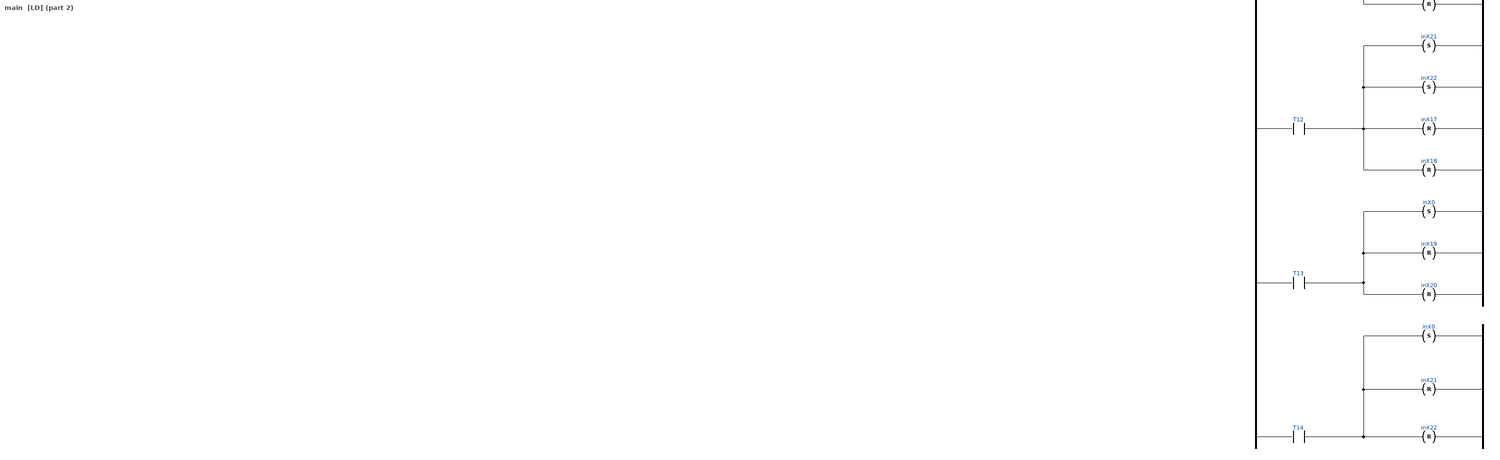
IF T12 THEN inX18 := FALSE; END_IF;
IF T12 THEN inX21 := TRUE; END_IF;
IF T12 THEN inX17 := FALSE; END_IF;
IF T12 THEN inX22 := TRUE; END_IF;
IF T13 THEN inX0 := TRUE; END_IF;
IF T13 THEN inX19 := FALSE; END_IF;
IF T13 THEN inX20 := FALSE; END_IF;
IF T14 THEN inX0 := TRUE; END_IF;
IF T14 THEN inX21 := FALSE; END_IF;
IF T14 THEN inX22 := FALSE; END_IF;
start := termX0;
_AND266_OUT := termX1 AND termX2 AND termX3;
WebGuide := _AND266_OUT;
CoilCar := _AND266_OUT;
Unwind := _AND266_OUT;
TensionSetup := termX4;
_AND271_OUT := termX5 AND termX6;
BottomKnife := _AND271_OUT;
TopKnife := _AND271_OUT;
_AND274_OUT := termX7 AND termX8;
MainDrive := _AND274_OUT;
PinchRoll := _AND274_OUT;
_AND277_OUT := termX9 AND termX10;
SlitWind := _AND277_OUT;
CoreShaft := _AND277_OUT;
_AND280_OUT := termX11 AND termX12;
NotchEdge := _AND280_OUT;
NotchUnwind := _AND280_OUT;
Press := termX15;
LaserSensor := termX16;
_AND287_OUT := termX19 AND termX20;
UnloadConv := _AND287_OUT;
Stack := _AND287_OUT;
_AND288_OUT := termX21 AND termX22;
RejConv := _AND288_OUT;
RejGate := _AND288_OUT;
BernoulliGenerator0(in := termX13 AND termX14, seed := seed_0);
Mechanical := BernoulliGenerator0.out_1;
Accum := BernoulliGenerator0.out_1 OR BernoulliGenerator0.out_2;
Laser := BernoulliGenerator0.out_2;
BernoulliGenerator1(in := termX17 AND termX18, seed := seed_1);
ElectrodePass := BernoulliGenerator1.out_1;
Vision := BernoulliGenerator1.out_1 OR BernoulliGenerator1.out_2;
ElectrodePass := NOT BernoulliGenerator1.out_2;
Dancer := BernoulliGenerator0.out_1 OR BernoulliGenerator0.out_2;
OQCConv := BernoulliGenerator1.out_1 OR BernoulliGenerator1.out_2;
END_PROGRAM

PROGRAM main2
  VAR
    inX0 : BOOL := TRUE;
    inX1 : BOOL;
    inX2 : BOOL;
    inX3 : BOOL;
    inX4 : BOOL;
    inX5 : BOOL;
    inX6 : BOOL;
    inX7 : BOOL;
    inX8 : BOOL;
    inX9 : BOOL;
    inX10 : BOOL;
    inX11 : BOOL;
    inX12 : BOOL;
    inX13 : BOOL;
    inX14 : BOOL;
    inX15 : BOOL;
    outX0 : BOOL;
    outX1 : BOOL;
    outX2 : BOOL;
    outX3 : BOOL;
    outX4 : BOOL;
    outX5 : BOOL;
    outX6 : BOOL;
    outX7 : BOOL;
    outX8 : BOOL;
    outX9 : BOOL;
    outX10 : BOOL;
    outX11 : BOOL;
    outX12 : BOOL;
    outX13 : BOOL;
    outX14 : BOOL;
    outX15 : BOOL;
    signalX0 : REAL;
    signalX1 : REAL;
    signalX2 : REAL;
    signalX3 : REAL;
    signalX4 : REAL;
    signalX5 : REAL;
    signalX6 : REAL;
    signalX7 : REAL;
    signalX8 : REAL;
    signalX9 : REAL;
    signalX10 : REAL;
    signalX11 : REAL;
    signalX12 : REAL;
    signalX13 : REAL;
    signalX14 : REAL;
    signalX15 : REAL;
    T0 : BOOL;
    T1 : BOOL;
    T2 : BOOL;
    T3 : BOOL;
    T4 : BOOL;
    T5 : BOOL;
    T6 : BOOL;
    T7 : BOOL;
    start : BOOL;
    ConvWeb : BOOL;
    TensWeb : BOOL;
    ConvCoat : BOOL;
    TensCoat : BOOL;
    PumpCoat : BOOL;
    ValveCoat : BOOL;
    ConvLevel : BOOL;
    TensLevel : BOOL;
    TensDryB : BOOL;
    AirB : BOOL;
    Heater : BOOL;
    AirA : BOOL;
    ConvQC : BOOL;
    TensQC : BOOL;
    Reset : BOOL;
    termX0 : BOOL;
    termX1 : BOOL;
    termX2 : BOOL;
    termX3 : BOOL;
    termX4 : BOOL;
    termX5 : BOOL;
    termX6 : BOOL;
    termX7 : BOOL;
    termX8 : BOOL;
    termX9 : BOOL;
    termX10 : BOOL;
    termX11 : BOOL;
    termX12 : BOOL;
    termX13 : BOOL;
    termX14 : BOOL;
    termX15 : BOOL;
    PVG0 : ProcessVariationGeneratorX0;
    PVG1 : ProcessVariationGeneratorX1;
    PVG2 : ProcessVariationGeneratorX2;
    PVG3 : ProcessVariationGeneratorX3;
    PVG4 : ProcessVariationGeneratorX4;
    PVG5 : ProcessVariationGeneratorX5;
    PVG6 : ProcessVariationGeneratorX6;
    PVG7 : ProcessVariationGeneratorX7;
    PVG8 : ProcessVariationGeneratorX8;
    PVG9 : ProcessVariationGeneratorX9;
    PVG10 : ProcessVariationGeneratorX10;
    PVG11 : ProcessVariationGeneratorX11;
    PVG12 : ProcessVariationGeneratorX12;
    PVG13 : ProcessVariationGeneratorX13;
    PVG14 : ProcessVariationGeneratorX14;
    PVG15 : ProcessVariationGeneratorX15;
  END_VAR

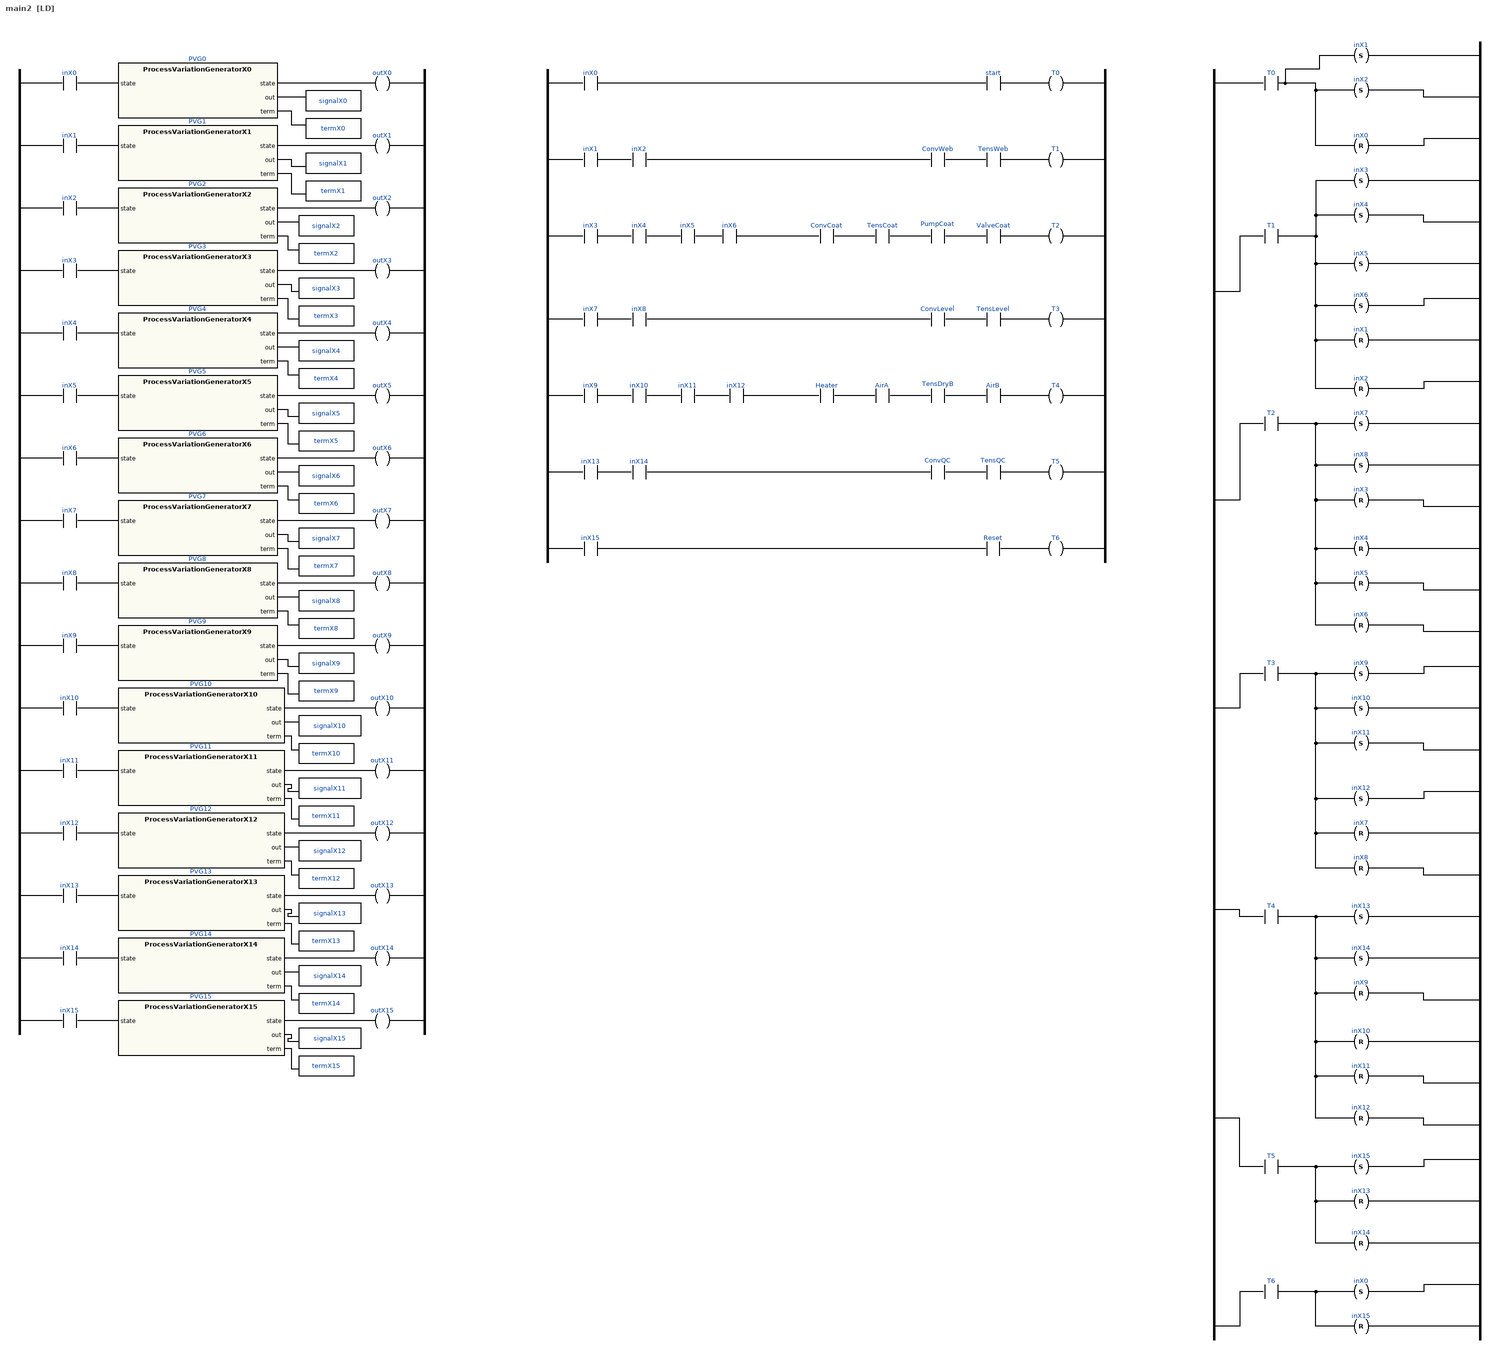
(* LD diagram, written out as Structured Text *)
PVG0(state := inX0);
outX0 := PVG0.state;
PVG1(state := inX1);
outX1 := PVG1.state;
PVG2(state := inX2);
outX2 := PVG2.state;
PVG3(state := inX3);
outX3 := PVG3.state;
PVG4(state := inX4);
outX4 := PVG4.state;
PVG5(state := inX5);
outX5 := PVG5.state;
PVG6(state := inX6);
outX6 := PVG6.state;
PVG7(state := inX7);
outX7 := PVG7.state;
PVG8(state := inX8);
outX8 := PVG8.state;
PVG9(state := inX9);
outX9 := PVG9.state;
PVG10(state := inX10);
outX10 := PVG10.state;
PVG11(state := inX11);
outX11 := PVG11.state;
PVG12(state := inX12);
outX12 := PVG12.state;
PVG13(state := inX13);
outX13 := PVG13.state;
PVG14(state := inX14);
outX14 := PVG14.state;
PVG15(state := inX15);
outX15 := PVG15.state;
signalX3 := PVG3.out;
signalX4 := PVG4.out;
signalX5 := PVG5.out;
signalX6 := PVG6.out;
signalX7 := PVG7.out;
signalX8 := PVG8.out;
signalX14 := PVG14.out;
signalX13 := PVG13.out;
signalX12 := PVG12.out;
signalX11 := PVG11.out;
signalX10 := PVG10.out;
signalX9 := PVG9.out;
signalX15 := PVG15.out;
signalX2 := PVG2.out;
signalX1 := PVG1.out;
signalX0 := PVG0.out;
T0 := inX0 AND start;
T1 := inX1 AND inX2 AND ConvWeb AND TensWeb;
T2 := inX3 AND inX4 AND inX5 AND inX6 AND ConvCoat AND TensCoat AND PumpCoat AND ValveCoat;
T3 := inX7 AND inX8 AND ConvLevel AND TensLevel;
T4 := inX9 AND inX10 AND inX11 AND inX12 AND Heater AND AirA AND TensDryB AND AirB;
T5 := inX13 AND inX14 AND ConvQC AND TensQC;
T6 := inX15 AND Reset;
IF T0 THEN inX1 := TRUE; END_IF;
IF T0 THEN inX2 := TRUE; END_IF;
IF T0 THEN inX0 := FALSE; END_IF;
IF T1 THEN inX3 := TRUE; END_IF;
IF T1 THEN inX4 := TRUE; END_IF;
IF T1 THEN inX5 := TRUE; END_IF;
IF T1 THEN inX6 := TRUE; END_IF;
IF T1 THEN inX1 := FALSE; END_IF;
IF T1 THEN inX2 := FALSE; END_IF;
IF T2 THEN inX8 := TRUE; END_IF;
IF T2 THEN inX3 := FALSE; END_IF;
IF T2 THEN inX4 := FALSE; END_IF;
IF T2 THEN inX5 := FALSE; END_IF;
IF T2 THEN inX6 := FALSE; END_IF;
IF T2 THEN inX7 := TRUE; END_IF;
IF T3 THEN inX9 := TRUE; END_IF;
IF T3 THEN inX10 := TRUE; END_IF;
IF T3 THEN inX11 := TRUE; END_IF;
IF T3 THEN inX12 := TRUE; END_IF;
IF T3 THEN inX7 := FALSE; END_IF;
IF T3 THEN inX8 := FALSE; END_IF;
IF T4 THEN inX13 := TRUE; END_IF;
IF T4 THEN inX14 := TRUE; END_IF;
IF T5 THEN inX13 := FALSE; END_IF;
IF T5 THEN inX14 := FALSE; END_IF;
IF T6 THEN inX0 := TRUE; END_IF;
IF T6 THEN inX15 := FALSE; END_IF;
IF T4 THEN inX9 := FALSE; END_IF;
IF T4 THEN inX10 := FALSE; END_IF;
IF T4 THEN inX11 := FALSE; END_IF;
IF T4 THEN inX12 := FALSE; END_IF;
IF T5 THEN inX15 := TRUE; END_IF;
termX15 := PVG15.term;
termX7 := PVG7.term;
termX0 := PVG0.term;
termX1 := PVG1.term;
termX2 := PVG2.term;
termX3 := PVG3.term;
termX4 := PVG4.term;
termX5 := PVG5.term;
termX12 := PVG12.term;
termX13 := PVG13.term;
termX11 := PVG11.term;
termX14 := PVG14.term;
termX10 := PVG10.term;
termX9 := PVG9.term;
termX8 := PVG8.term;
termX6 := PVG6.term;
END_PROGRAM

CONFIGURATION Config0
  RESOURCE Res0 ON PLC
    TASK task0(INTERVAL := T#20ms, PRIORITY := 0);
    PROGRAM instance0 WITH task0 : main;
  END_RESOURCE
END_CONFIGURATION
